INTERFACE ITcoAnalogueInspector

(*~
<docu>
<summary>
	Inspects the signal and evaluates that it matches the value set in `RequiredStatus`.
</summary>
<returns>
	Returns the interface with information about the state of inspection.
</returns>
</docu>
~*)
METHOD Inspect : IInspector
VAR_INPUT
    Status : LREAL;
END_VAR
END_METHOD

END_INTERFACE

(* stored: Version 1.1.0.1, ProductVersion 3.1.4024.9
   Itf ITcoAnalogueInspector: Id {7df2cfa4-e810-05a2-2931-9dc354df0c62}
   Method Inspect: Id {fa878bf0-8f5f-03f6-3b75-ba33769e65e0} *)
